// TIA Portal V20 export
TYPE "typeAxisHomeCondition"
// stored: Access Published, Namespace LER
   STRUCT
      HomeInterlock : Bool;
      homeinterlock_error : Bool;
      intout : Array[0..9] of Bool;
   END_STRUCT;
END_TYPE
